// TwinCAT 3 PLC project SampleWeighing
// ProgramVersion: 3.1.4026.20
// libraries:
//   Tc2_Standard, * (Beckhoff Automation GmbH)
//   Tc2_SUPS, * (Beckhoff Automation GmbH)
//   Tc2_System, * (Beckhoff Automation GmbH)
//   Tc2_Utilities, * (Beckhoff Automation GmbH)
//   Tc3_EventLogger, * (Beckhoff Automation GmbH)
//   Tc3_Filter, * (Beckhoff Automation GmbH)
//   Tc3_Module, * (Beckhoff Automation GmbH)
//   Tc3_Weighing, * (Beckhoff Automation GmbH)
// project tree:
//   DUTs/ E_DistributionType.TcDUT (not stored), E_FilterType.TcDUT, E_FunctionType.TcDUT, ST_POINTS.TcDUT
//   GVLs/ Global_Constants.TcGVL, GVL_IO.TcGVL, GVL_WEIGHING_HMI.TcGVL
//   / PlcTask.TcTTO
//   POUs/FBs/ FB_CLOCK.TcPOU (not stored), FB_Filter.TcPOU, FB_Filter59.TcPOU, P_TextModeWrite.TcPOU
//   POUs/ FB_DynamicWeighing.TcPOU, FB_STATS.TcPOU, MAIN.TcPOU, P_HMI.TcPOU, P_LightTest.TcPOU (not stored)
//   POUs/Utilities/ FB_FunctionGenerator.TcPOU
//   VISUs/ RecipeManager.TcRMO (not stored)
// real-time tasks:
//   TASK PlcTask: cycle T#1ms, priority 4, ADS port 350
// I/O:
//   DEVICE Device 2 (EtherCAT), AmsNetId 10.199.162.27.3.1
//     Term 1 (EK1100) [EK1100 EtherCAT Coupler (2A E-Bus)]
//       Term 2 (EL1809) [EL1809 16Ch. Dig. Input 24V, 3ms]
//       Term 3 (EL2808) [EL2808 8Ch. Dig. Output 24V, 0.5A]
//       Term 5 (EL4132)
//       Term 10 (EL9510) [EL9510 Power supply terminal 10V]
//       Term 11 (EL3102) [EL3102 2Ch. Ana. Input +/-10V, Diff.]
//       Term 16 (EL6751) [EL6751 CANopen Master]
//       Term 9 (EL9011) [EL9011 End Terminal]
//     Term 14 (EK1100) [EK1100 EtherCAT Coupler (2A E-Bus)]
//       Term 15 (EL3356-0010) [EL3356-0010 1Ch. Ana. Input Resistor Bridge Terminal, 24bit, High Precision]
//       Term 12 (EL3356) [EL3356 1Ch. Ana. Input Resistor Bridge Terminal, 16bit, High Precision]
//       Term 20 (EK1110) [EK1110 EtherCAT extension]
// variable links:
//   SampleWeighing/SampleWeighing Instance <-> Device 2 (EtherCAT)/Term 1 (EK1100)/Term 2 (EL1809)
//     PlcTask Inputs/GVL_IO.arrDIs[{1..16}] <-> Channel {1..16}/Input  (16 links)
//   SampleWeighing/SampleWeighing Instance <-> Device 2 (EtherCAT)/Term 1 (EK1100)/Term 3 (EL2808)
//     PlcTask Outputs/GVL_IO.arrDOs[{1..8}] <-> Channel {1..8}/Output  (8 links)
//   SampleWeighing/SampleWeighing Instance <-> Device 2 (EtherCAT)/Term 1 (EK1100)/Term 5 (EL4132)
//     PlcTask Outputs/GVL_IO.arrAOs[1] <-> Channel 1/Output
//     PlcTask Outputs/GVL_IO.arrAOs[2] <-> Channel 2/Output
//   SampleWeighing/SampleWeighing Instance <-> Device 2 (EtherCAT)/Term 14 (EK1100)/Term 15 (EL3356-0010)
//     PlcTask Inputs/GVL_IO.EL3356_RawInput <-> RMB Value (Real)/Value (Real)
//     PlcTask Outputs/GVL_IO.EL3356_SampleMode <-> RMB Control/Ctrl/Sample mode

CONFIGURATION SampleWeighing
    RESOURCE PLC ON TwinCAT3
        TASK PlcTask(INTERVAL := T#1ms, PRIORITY := 4);
        PROGRAM MAIN WITH PlcTask : MAIN;
    END_RESOURCE
END_CONFIGURATION

// ---- DUTs/E_FilterType.TcDUT
{attribute 'qualified_only'}
{attribute 'strict'}
{attribute 'to_string'}
TYPE E_FilterType :
(	
	Disabled := 0,
	PTn,
	MovingAverage
);
END_TYPE

// ---- DUTs/E_FunctionType.TcDUT
TYPE E_FunctionType :
(
	eConst := 0,
	eSine,
	eSquare,
	ePulse,
	eTriangular,
	eSawtooth,
	eAM,
	eRand,
	eTrapezoid
);
END_TYPE

// ---- DUTs/ST_POINTS.TcDUT
TYPE ST_POINTS :
STRUCT
	x : REAL;
	y : REAL;
END_STRUCT
END_TYPE

// ---- GVLs/Global_Constants.TcGVL
VAR_GLOBAL CONSTANT
	cOversamples	: UINT := 1;					// number of oversamples
	cSamplingRate	: UINT := 1000 * cOversamples;	// samplerate
END_VAR

// ---- GVLs/GVL_IO.TcGVL
{attribute 'qualified_only'}
VAR_GLOBAL
	arrDIs				 		AT %I*	: ARRAY[1..16] OF BOOL;
	arrDOs			 			AT %Q*	: ARRAY[1..8] OF BOOL;
	arrAIs						AT %I*	: ARRAY[1..2] OF INT;
	arrAOs						AT %Q*	: ARRAY[1..2] OF INT;
	EL3356_RawInput 			AT %I*	: REAL;
	EL3356_SampleMode			AT %Q*	: BOOL := FALSE;
END_VAR

// ---- GVLs/GVL_WEIGHING_HMI.TcGVL
{attribute 'qualified_only'}
VAR_GLOBAL PERSISTENT
	(* Combo Filter Cfg *)
	nFilterOrder 		: UINT := 6;
	rCutOff		 		: REAL	:= 10.0;
	cSamplingRate		: UINT := 100 * cOversamples;	// samplerate
	nSamplesToFilter	: UINT := 200;
	bResetFilter		: BOOL;
	fNotchFrequency		: LREAL;
	
	(* Scaling Params *)
	fRawLow 				: REAL := 0.0;
	fReferenceLow 			: REAL := 0.0;
	fRawHigh 				: REAL := 1000.0;
	fReferenceHigh 			: REAL := 100.0;
	nNumCalibrationSamples 	: UDINT := 100;
	
	(* Weighing Params *)
	nWindowLenght 					: UDINT := 100;
	
	nValidationSamplesValidation	: UDINT := 100;
	fThresholdWeightValidation 		: LREAL := 20.0;
	fMaxStdValidation				: LREAL := 5.0;
	fMaxWeightDeviationValidation	: LREAL := 0.0;
	fRelativeWeightLimit			: LREAL := 0.0;
	fActualRelativeWeightLimit		: LREAL := 0.0;
	
	
	nValidationSamplesAutoTare		: UDINT := 100;
	fThresholdWeightAutoTare 		: REAL := 10.0;
	fMaxStdAutoTare					: LREAL := 1.0;
	fMaxWeightDeviationAutoTare		: LREAL := 0.0;
	
		
	(* Booleans to Reconfigure Filters By IHM *)
	bReconfigureFilter 		: BOOL;
	bReconfigureWeighing 	: BOOL;
	
	(* Calibration *)
	fCalibrateReferenceLow 		: LREAL := 0;
	fCalibrateReferenceHigh 	: LREAL := 1000;
	bCalibrateReferenceLow 		: BOOL := FALSE;
	bCalibrateReferenceHigh 	: BOOL := FALSE;
	bApplyCalibration 			: BOOL := FALSE;
	bAcceptCalibration 			: BOOL := TRUE;
	
	(* Tare *)	
	bTare : BOOL := FALSE;
	fMaxTotalTareLimit : LREAL := 40.0; // set error if total taring amount exceeds the limit
	eAutoTareType : E_WG_AutoTareType := E_WG_AutoTareType.eContinously;
	nNumTareSamples 		: UDINT := 100;
	
	(* Filters Cfg *)	
	
	EFilter1			: E_FilterType;
	EFilter2			: E_FilterType;
	EFilter3			: E_FilterType;
	EFilter4			: E_FilterType;
	EFilter5			: E_FilterType;
	
	(* Filter 1 *)
	fc1				 	: LREAL := 3; // Cut Frequency in Hz
	Tfc1			 	: LREAL := (1.0 / (2.0 * PI * fc1)) / SQRT(EXPT(2.0, 1.0 / 1) - 1.0);
	nGainPTn1			: UINT := 1;
	nOrderPTn1			: UINT := 1;
	fSamplingRatePTn1	: UINT := 1000;
	bReconfigurePTn1	: BOOL;
	
	STFilter1_PTn		: ST_FTR_PTn := (fKp:= 1,
										 fT1 := Tfc1,
										 nOrder := nOrderPTn1,
										 fSamplingRate := fSamplingRatePTn1,
										 nOversamples:= 1,
										 nChannels := 1);
	
	fbFilterPTn1 : FB_FTR_PTn := (stConfig:= STFilter1_PTn);
	
	(* Filter 2 *)
	fc2                  : LREAL := 3;
	Tfc2                 : LREAL := (1.0 / (2.0 * PI * fc2)) / SQRT(EXPT(2.0, 1.0 / 1) - 1.0);
	nGainPTn2            : UINT := 1;
	nOrderPTn2           : UINT := 1;
	fSamplingRatePTn2    : UINT := 1000;
	bReconfigurePTn2     : BOOL;
	
	STFilter2_PTn        : ST_FTR_PTn := (
							fKp:= 1,
							fT1 := Tfc2,
							nOrder := nOrderPTn2,
							fSamplingRate := fSamplingRatePTn2,
							nOversamples:= 1,
							nChannels := 1);
	
	fbFilterPTn2 : FB_FTR_PTn := (stConfig:= STFilter2_PTn);
	
	(* Filter 3 *)
	fc3                  : LREAL := 3;
	Tfc3                 : LREAL := (1.0 / (2.0 * PI * fc3)) / SQRT(EXPT(2.0, 1.0 / 1) - 1.0);
	nGainPTn3            : UINT := 1;
	nOrderPTn3           : UINT := 1;
	fSamplingRatePTn3    : UINT := 1000;
	bReconfigurePTn3     : BOOL;
	
	STFilter3_PTn        : ST_FTR_PTn := (
							fKp:= 1,
							fT1 := Tfc3,
							nOrder := nOrderPTn3,
							fSamplingRate := fSamplingRatePTn3,
							nOversamples:= 1,
							nChannels := 1);
	
	fbFilterPTn3 : FB_FTR_PTn := (stConfig:= STFilter3_PTn);
	
	(* Filter 4 *)
	fc4                  : LREAL := 3;
	Tfc4                 : LREAL := (1.0 / (2.0 * PI * fc4)) / SQRT(EXPT(2.0, 1.0 / 1) - 1.0);
	nGainPTn4            : UINT := 1;
	nOrderPTn4           : UINT := 1;
	fSamplingRatePTn4    : UINT := 1000;
	bReconfigurePTn4     : BOOL;
	
	STFilter4_PTn        : ST_FTR_PTn := (
							fKp:= 1,
							fT1 := Tfc4,
							nOrder := nOrderPTn4,
							fSamplingRate := fSamplingRatePTn4,
							nOversamples:= 1,
							nChannels := 1);
	
	fbFilterPTn4 : FB_FTR_PTn := (stConfig:= STFilter4_PTn);
	
	(* Filter 5 *)
	fc5                  : LREAL := 3;
	Tfc5                 : LREAL := (1.0 / (2.0 * PI * fc5)) / SQRT(EXPT(2.0, 1.0 / 1) - 1.0);
	nGainPTn5            : UINT := 1;
	nOrderPTn5           : UINT := 1;
	fSamplingRatePTn5    : UINT := 1000;
	bReconfigurePTn5     : BOOL;
	
	STFilter5_PTn        : ST_FTR_PTn := (
							fKp:= 1,
							fT1 := Tfc5,
							nOrder := nOrderPTn5,
							fSamplingRate := fSamplingRatePTn5,
							nOversamples:= 1,
							nChannels := 1);
	
	fbFilterPTn5 : FB_FTR_PTn := (stConfig:= STFilter5_PTn);
	
	(* Mirror actual values to simplify to user *)
	(* Validation *)
	nActualWindowLenght 					: UDINT;
	nActualValidationSamplesValidation		: UDINT;
	fActualThresholdWeightValidation 		: LREAL;
	fActualMaxStdValidation					: LREAL;
	fActualMaxWeightDeviationValidation		: LREAL;
	
	(* Last and Actual Weigh Values *)
	fWeight 		: LREAL;
	fLastWeight 	: LREAL;
	fStd 			: LREAL;
	fLastStd 		: LREAL;
	
	(* Lib Booleans *)
	bValidMeasurement 	: BOOL;
	bNewResult			: BOOL;
	bCriteria1			: BOOL;
	bCriteria2			: BOOL;
	bCriteria3			: BOOL;
	
	
END_VAR

// ---- POUs/MAIN.TcPOU
PROGRAM MAIN
VAR
	// Test signal generation
	fRawAmplitudeSignal 	: LREAL := 1000;
	fAbsoluteNoise 			: LREAL := 200;
	fFrequency 				: LREAL := 1; 			// Hz		
	fSamplingRate 			: LREAL := TO_LREAL(cSamplingRate);
	fbSignal 				: FB_FunctionGenerator;
	
	aRawInput 				: ARRAY[1..cOversamples] OF LREAL;
	aRawInputNoise 			: ARRAY[1..cOversamples] OF LREAL;	
	aRawSignal	 			: ARRAY[1..cOversamples] OF LREAL;
	
	// Error handling
	nCountErrors 			: UDINT;
	nEventId 				: UDINT;
	sEventClassName 		: T_MaxString;
	sSourcePath 			: T_MaxString;
	eSeverity 				: TcEventSeverity;
	
	// Weighing
	fbDynamicWeighing 		: FB_DynamicWeighing;
	
	
	//Slope
	bActivateSlope 			: BOOL;
	fDeltaWeight 			: LREAL;
	bAddWeight				: BOOL;
	
	// CP67 UPS Persistent Data
	fbUPS				: FB_S_UPS_BAPI;
	
	stParamsFilterIn 	: ST_WG_ComboFilter;
	stParamsScaleIn		: ST_WG_Scaling;
	stParamsWeighingIn	: ST_WG_Weighing;
	
	bInit				: BOOL;
	bSuccess			: BOOL;
	yFiltroEntrada		: LREAL;
	yFiltroSaida		: LREAL;
	yFiltroSaida2		: LREAL;
	yFiltroSaida3		: LREAL;
	yFiltroSaida4		: LREAL;
	yFiltroSaida5		: LREAL;
				
	bSucceed			: BOOL;
	bReset: BOOL;
END_VAR

// Generate inputs FOR simulation
GenerateInputs();

// Increase the weight continuously.
IF bActivateSlope THEN
	AddSlope();
END_IF

// Increase the weight once
IF bAddWeight THEN
	AddWeight();
	bAddWeight := FALSE;
END_IF

// // Call weighing FB
// fbDynamicWeighing(aInput := aRawInputNoise);

actFilterCfg();
actFilterSignal();

(* Filter Params *)
stParamsFilterIn.nOrder 			:= GVL_WEIGHING_HMI.nFilterOrder;
stParamsFilterIn.fCutoff 			:= GVL_WEIGHING_HMI.rCutOff;
stParamsFilterIn.fSamplingRate 		:= TO_LREAL(GVL_WEIGHING_HMI.cSamplingRate);
stParamsFilterIn.nSamplesToFilter 	:= GVL_WEIGHING_HMI.nSamplesToFilter;
stParamsFilterIn.bReset				:= GVL_WEIGHING_HMI.bResetFilter;
stParamsFilterIn.fNotchFrequency	:= GVL_WEIGHING_HMI.fNotchFrequency;


(* Scale Params *)
stParamsScaleIn.fRawLow 				:= GVL_WEIGHING_HMI.fRawLow;
stParamsScaleIn.fReferenceLow 			:= GVL_WEIGHING_HMI.fReferenceLow;
stParamsScaleIn.fRawHigh		 		:= GVL_WEIGHING_HMI.fRawHigh;
stParamsScaleIn.fReferenceHigh			:= GVL_WEIGHING_HMI.fReferenceHigh;


(* Weighing *)
stParamsWeighingIn.nWindowLength						:= GVL_WEIGHING_HMI.nWindowLenght;
stParamsWeighingIn.Validation.nValidationSamples		:= GVL_WEIGHING_HMI.nValidationSamplesValidation;
stParamsWeighingIn.Validation.fThresholdWeight			:= GVL_WEIGHING_HMI.fThresholdWeightValidation;
stParamsWeighingIn.Validation.fMaxStd					:= GVL_WEIGHING_HMI.fMaxStdValidation;
stParamsWeighingIn.Validation.fMaxWeightDeviation		:= GVL_WEIGHING_HMI.fMaxWeightDeviationValidation;
stParamsWeighingIn.Validation.fRelativeWeightLimit		:= GVL_WEIGHING_HMI.fRelativeWeightLimit;


stParamsWeighingIn.AutoTare.nValidationSamples			:= GVL_WEIGHING_HMI.nValidationSamplesAutoTare;
stParamsWeighingIn.AutoTare.fThresholdWeight			:= GVL_WEIGHING_HMI.fThresholdWeightAutoTare;
stParamsWeighingIn.AutoTare.fMaxStd						:= GVL_WEIGHING_HMI.fMaxStdAutoTare;
stParamsWeighingIn.AutoTare.fMaxWeightDeviation			:= GVL_WEIGHING_HMI.fMaxWeightDeviationAutoTare;


(* Controls *)			  


fbDynamicWeighing(aInput := aRawSignal, 
					stParamsComboFilter 		:= stParamsFilterIn,
					stParamsScale 				:= stParamsScaleIn,
					stParamsWeighing 			:= stParamsWeighingIn,
					nNumCalibrationSamples 		:= GVL_WEIGHING_HMI.nNumCalibrationSamples,
					nNumTareSamples 			:= GVL_WEIGHING_HMI.nNumTareSamples,
					bAcceptCalibration			:= GVL_WEIGHING_HMI.bAcceptCalibration,
					fCalibrateReferenceLow 		:= GVL_WEIGHING_HMI.fCalibrateReferenceLow,
					fCalibrateReferenceHigh 	:= GVL_WEIGHING_HMI.fCalibrateReferenceHigh,
					bTare						:= GVL_WEIGHING_HMI.bTare,
					fMaxTotalTareLimit			:= GVL_WEIGHING_HMI.fMaxTotalTareLimit,
					eAutoTareType				:= GVL_WEIGHING_HMI.eAutoTareType,
);
	
// Error handling
IF fbDynamicWeighing.ipResultMessage <> 0 THEN	
	nEventId := fbDynamicWeighing.ipResultMessage.nEventId;
	sSourcePath := fbDynamicWeighing.ipResultMessage.ipSourceInfo.sName;
	eSeverity := fbDynamicWeighing.ipResultMessage.eSeverity;	
	fbDynamicWeighing.ipResultMessage.RequestEventClassName(1033, sEventClassName, SIZEOF(sEventClassName));
END_IF

IF fbDynamicWeighing.bError THEN
	nCountErrors := nCountErrors + 1;
END_IF


(* HMI Mirroring important variables to user *)
P_HMI();


(* CSV Export *)
//P_TextModeWrite.database();

ACTION actAux:
(* Light Test *)
P_LightTest();

(* HMI *)
P_HMI();

(* UPS *)
fbUPS(
	sNetID:= '', 
	iPLCPort:= 851, 
	tTimeout:= , 
	eUpsMode:= , 
	ePersistentMode:= , 
	tRecoverTime:= , 
	bPowerFailDetect=> , 
	eState=> , 
	nCapacity=> , 
	bBusy=> , 
	bError=> , 
	nErrID=> );
END_ACTION

ACTION actFilterCfg:
IF GVL_WEIGHING_HMI.bReconfigurePTn1 THEN
	GVL_WEIGHING_HMI.STFilter1_PTn.fKp 				:= GVL_WEIGHING_HMI.nGainPTn1;
	GVL_WEIGHING_HMI.STFilter1_PTn.fT1 				:= GVL_WEIGHING_HMI.Tfc1;
	GVL_WEIGHING_HMI.STFilter1_PTn.nOrder 			:= GVL_WEIGHING_HMI.nOrderPTn1;
	GVL_WEIGHING_HMI.STFilter1_PTn.fSamplingRate 	:= GVL_WEIGHING_HMI.fSamplingRatePTn1;
	GVL_WEIGHING_HMI.STFilter1_PTn.nOversamples		:= 1;
	GVL_WEIGHING_HMI.STFilter1_PTn.nChannels 		:= 1;	

	bSuccess := GVL_WEIGHING_HMI.fbFilterPTn1.Configure(stConfig:=GVL_WEIGHING_HMI.STFilter1_PTn);
END_IF


IF bReset THEN
	GVL_WEIGHING_HMI.fbFilterPTn1.Reset();
END_IF


IF GVL_WEIGHING_HMI.bReconfigurePTn2 THEN
	GVL_WEIGHING_HMI.STFilter2_PTn.fKp 				:= GVL_WEIGHING_HMI.nGainPTn2;
	GVL_WEIGHING_HMI.STFilter2_PTn.fT1 				:= GVL_WEIGHING_HMI.Tfc2;
	GVL_WEIGHING_HMI.STFilter2_PTn.nOrder 			:= GVL_WEIGHING_HMI.nOrderPTn2;
	GVL_WEIGHING_HMI.STFilter2_PTn.fSamplingRate 	:= GVL_WEIGHING_HMI.fSamplingRatePTn2;
	GVL_WEIGHING_HMI.STFilter2_PTn.nOversamples		:= 1;
	GVL_WEIGHING_HMI.STFilter2_PTn.nChannels 		:= 1;	

	bSuccess := GVL_WEIGHING_HMI.fbFilterPTn2.Configure(stConfig:=GVL_WEIGHING_HMI.STFilter2_PTn);
END_IF

IF GVL_WEIGHING_HMI.bReconfigurePTn3 THEN
	GVL_WEIGHING_HMI.STFilter3_PTn.fKp 				:= GVL_WEIGHING_HMI.nGainPTn3;
	GVL_WEIGHING_HMI.STFilter3_PTn.fT1 				:= GVL_WEIGHING_HMI.Tfc3;
	GVL_WEIGHING_HMI.STFilter3_PTn.nOrder 			:= GVL_WEIGHING_HMI.nOrderPTn3;
	GVL_WEIGHING_HMI.STFilter3_PTn.fSamplingRate 	:= GVL_WEIGHING_HMI.fSamplingRatePTn3;
	GVL_WEIGHING_HMI.STFilter3_PTn.nOversamples		:= 1;
	GVL_WEIGHING_HMI.STFilter3_PTn.nChannels 		:= 1;	

	bSuccess := GVL_WEIGHING_HMI.fbFilterPTn3.Configure(stConfig:=GVL_WEIGHING_HMI.STFilter3_PTn);
END_IF


IF GVL_WEIGHING_HMI.bReconfigurePTn4 THEN
	GVL_WEIGHING_HMI.STFilter4_PTn.fKp 				:= GVL_WEIGHING_HMI.nGainPTn4;
	GVL_WEIGHING_HMI.STFilter4_PTn.fT1 				:= GVL_WEIGHING_HMI.Tfc4;
	GVL_WEIGHING_HMI.STFilter4_PTn.nOrder 			:= GVL_WEIGHING_HMI.nOrderPTn4;
	GVL_WEIGHING_HMI.STFilter4_PTn.fSamplingRate 	:= GVL_WEIGHING_HMI.fSamplingRatePTn4;
	GVL_WEIGHING_HMI.STFilter4_PTn.nOversamples		:= 1;
	GVL_WEIGHING_HMI.STFilter4_PTn.nChannels 		:= 1;	

	bSuccess := GVL_WEIGHING_HMI.fbFilterPTn4.Configure(stConfig:=GVL_WEIGHING_HMI.STFilter4_PTn);
END_IF


IF GVL_WEIGHING_HMI.bReconfigurePTn5 THEN
	GVL_WEIGHING_HMI.STFilter5_PTn.fKp 				:= GVL_WEIGHING_HMI.nGainPTn5;
	GVL_WEIGHING_HMI.STFilter5_PTn.fT1 				:= GVL_WEIGHING_HMI.Tfc5;
	GVL_WEIGHING_HMI.STFilter5_PTn.nOrder 			:= GVL_WEIGHING_HMI.nOrderPTn5;
	GVL_WEIGHING_HMI.STFilter5_PTn.fSamplingRate 	:= GVL_WEIGHING_HMI.fSamplingRatePTn5;
	GVL_WEIGHING_HMI.STFilter5_PTn.nOversamples		:= 1;
	GVL_WEIGHING_HMI.STFilter5_PTn.nChannels 		:= 1;	

	bSuccess := GVL_WEIGHING_HMI.fbFilterPTn5.Configure(stConfig:=GVL_WEIGHING_HMI.STFilter5_PTn);
END_IF
END_ACTION

ACTION actFilterSignal:
// aRawSignal[1] := GVL_IO.EL3356_RawInput;

// yFiltroEntrada := GVL_IO.EL3356_RawInput;

yFiltroEntrada := aRawInputNoise[1];

(* First Filter *)
IF GVL_WEIGHING_HMI.EFilter1 = 0 THEN // Disabled
	yFiltroSaida := yFiltroEntrada;	
ELSIF GVL_WEIGHING_HMI.EFilter1 = 1 THEN // PTn
	bSucceed := GVL_WEIGHING_HMI.fbFilterPTn1.Call(ADR(yFiltroEntrada), SIZEOF(yFiltroEntrada), ADR(yFiltroSaida), SIZEOF(yFiltroSaida));
END_IF

(* Second Filter *)
IF GVL_WEIGHING_HMI.EFilter2 = 0 THEN // Disabled
	yFiltroSaida2 := yFiltroSaida;	
ELSIF GVL_WEIGHING_HMI.EFilter2 = 1 THEN // PTn
	bSucceed := GVL_WEIGHING_HMI.fbFilterPTn2.Call(ADR(yFiltroSaida), SIZEOF(yFiltroSaida), ADR(yFiltroSaida2), SIZEOF(yFiltroSaida2));
END_IF

(* Third Filter *)
IF GVL_WEIGHING_HMI.EFilter3 = 0 THEN // Disabled
	yFiltroSaida3 := yFiltroSaida2;	
ELSIF GVL_WEIGHING_HMI.EFilter3 = 1 THEN // PTn
	bSucceed := GVL_WEIGHING_HMI.fbFilterPTn2.Call(ADR(yFiltroSaida2), SIZEOF(yFiltroSaida2), ADR(yFiltroSaida3), SIZEOF(yFiltroSaida3));
END_IF

(* Fourth Filter *)
IF GVL_WEIGHING_HMI.EFilter4 = 0 THEN // Disabled
	yFiltroSaida4 := yFiltroSaida3;	
ELSIF GVL_WEIGHING_HMI.EFilter4 = 1 THEN // PTn
	bSucceed := GVL_WEIGHING_HMI.fbFilterPTn2.Call(ADR(yFiltroSaida3), SIZEOF(yFiltroSaida3), ADR(yFiltroSaida4), SIZEOF(yFiltroSaida4));
END_IF

(* Fifth Filter *)
IF GVL_WEIGHING_HMI.EFilter5 = 0 THEN // Disabled
	yFiltroSaida5 := yFiltroSaida4;	
ELSIF GVL_WEIGHING_HMI.EFilter5 = 1 THEN // PTn
	bSucceed := GVL_WEIGHING_HMI.fbFilterPTn2.Call(ADR(yFiltroSaida4), SIZEOF(yFiltroSaida4), ADR(yFiltroSaida5), SIZEOF(yFiltroSaida5));
END_IF


aRawSignal[1] := yFiltroSaida5; // Recebe sempre a última saída
END_ACTION

METHOD AddSlope : BOOL
VAR_INPUT
END_VAR
VAR
	idx : UINT;
	fSlope: LREAL := 0.2;
END_VAR
fDeltaWeight := fDeltaWeight + fSlope;
END_METHOD

METHOD AddWeight : BOOL
VAR_INPUT
END_VAR
VAR
	idx : UINT;
	fAddWeight: LREAL := 100;
END_VAR
fDeltaWeight := fDeltaWeight + fAddWeight;
END_METHOD

METHOD GenerateInputs : BOOL
VAR_INPUT
END_VAR
VAR
	idx : UINT;
END_VAR
fbSignal(				
	fSamplingRate := fSamplingRate,
	nOversamples := cOversamples,
	fFrequency := fFrequency,
	fAmplitude := 2.0 * fRawAmplitudeSignal,
	eFunction := E_FunctionType.eTrapezoid,							
	aSignal => aRawInput);


FOR idx := 1 TO cOversamples DO
	aRawInput[idx] := aRawInput[idx] + fDeltaWeight;
END_FOR		 

MEMCPY(ADR(aRawInputNoise),ADR(aRawInput),SIZEOF(aRawInputNoise));
fbSignal.AddAbsoluteNoise(fAbsoluteNoise, aRawInputNoise);
END_METHOD

END_PROGRAM

// ---- POUs/Utilities/FB_FunctionGenerator.TcPOU
// generates a signal build up by the specified function type. v1.4
// generates random signal (uniform, normal or chi-squared)

FUNCTION_BLOCK FB_FunctionGenerator
VAR_INPUT
	bEnable		: BOOL 	:= TRUE;
	fSamplingRate : LREAL := 10000.0; // in Hz
	nOversamples : UDINT := 10;
	fFrequency	: LREAL := 1000;	// in [Hz]
	fAmplitude	: LREAL := 1;
	fOffset		: LREAL	:= 0;	
	nDutyCycle	: UINT 	:= 50;		// % (for pulse function)
	nSeed		: INT	:= 1;	 
	aRange		: ARRAY [1..2] OF LREAL := [0,1];
	eRandType	: E_DistributionType	:= E_DistributionType.eNormal;
	eFunction	: E_FunctionType := E_FunctionType.eSine;	
END_VAR
VAR_OUTPUT
	bError		: BOOL;
	aSignal		: ARRAY[1..cOversamples] OF LREAL;
END_VAR
VAR
	bInit						: BOOL := TRUE;
	fLastSamplingRate : LREAL;
	nLastOversamples : UDINT;
	fLastFrequency				: LREAL;		// in [Hz]
	fLastAmplitude				: LREAL;
	fLastOffset					: LREAL;
	nLastDutyCycle				: UINT;
	eLastFunction				: E_FunctionType;
	
	nSamples					: UDINT;
	fCycleTime					: LREAL;		// in [s]
	fDelta						: LREAL;		// amplitude delta per sample
	fPhase						: LREAL;		// in [°]
	nSign						: INT := 1;		// 1 or -1
	fLastSignalValue			: LREAL;		// amplitude
	fPeriod						: LREAL;		// in [s]
	fAngularIncrement			: LREAL;		// in [°]
	fAngularIncrementPerCycle	: LREAL;		// in [°]
	fAngularIncrementPerSample	: LREAL;		// in [°]
	(* for modulated signal *)
	fCarrierFrequency			: LREAL := 500;	// in [Hz] (sine)
	fCarrierAmplitude			: LREAL := 1;
	fCarrierPeriod				: LREAL;		// in [s]
	fCarrierAngularIncrement			: LREAL;		// in [°]
	fCarrierAngularIncrementPerCycle	: LREAL;		// in [°]
	fCarrierAngularIncrementPerSample	: LREAL;		// in [°]
	
	fbDrand						: ARRAY[1..cOversamples] OF DRAND;		
	bNormalDist					: BOOL := TRUE;
	
	fY1							: LREAL;
	fY2							: LREAL;
	fX1							: LREAL;
	fX2							: LREAL;
	
	fbRAND1						: DRAND;
	fbRAND2						: DRAND;				
END_VAR

IF bEnable THEN

	IF fLastSamplingRate <> fSamplingRate THEN
		bInit := TRUE; // For automatic initializing
		fLastSamplingRate := fSamplingRate;
	END_IF
	IF nLastOversamples <> nOversamples THEN
		bInit := TRUE; // For automatic initializing
		nLastOversamples := nOversamples;
	END_IF
	
	IF fLastFrequency <> fFrequency THEN
		bInit := TRUE; // For automatic initializing
		fLastFrequency := fFrequency;
	END_IF
	IF fLastAmplitude <> fAmplitude THEN
		bInit := TRUE; // For automatic initializing
		fLastAmplitude := fAmplitude;
	END_IF
	IF fLastOffset <> fOffset THEN
		bInit := TRUE; // For automatic initializing
		fLastOffset := fOffset;
	END_IF
	IF nLastDutyCycle <> nDutyCycle THEN
		bInit := TRUE; // For automatic initializing
		nLastDutyCycle := nDutyCycle;
	END_IF
	IF eLastFunction <> eFunction THEN
		bInit := TRUE; // For automatic initializing
		eLastFunction := eFunction;
	END_IF
	IF bInit THEN
		// Get taks info	
//		fbGetTaskIdx();
//		fCycleTime := TwinCAT_SystemInfoVarList._TaskInfo[fbGetTaskIdx.index].CycleTime (*100ns*) / (10.0 * 1000.0 * 1000.0);	
		fCycleTime	 := nOversamples/fSamplingRate;
		fLastSignalValue := 0;
		nSign := 1;
		fAngularIncrement := 0;
		// Flush out old data
		MEMSET(ADR(aSignal), 0, SIZEOF(aSignal));
		IF fFrequency <> 0 AND fCycleTime > 0 THEN		
			// Calculate period, increments per plc cycle, increment per oversample
			IF cOversamples <> 0 THEN			
				IF eFunction = E_FunctionType.eSine THEN
					fPeriod := 1/fFrequency;
					fAngularIncrementPerCycle := 360*(fCycleTime/fPeriod);
					fAngularIncrementPerSample := fAngularIncrementPerCycle/cOversamples;
					// no phase adjustment
					bInit := FALSE;
				ELSIF eFunction = E_FunctionType.eConst	THEN
					bInit := FALSE;	
				ELSIF eFunction = E_FunctionType.eSquare	THEN
					fPeriod := 1/fFrequency;
					fAngularIncrementPerCycle := 360*(fCycleTime/fPeriod);
					fAngularIncrementPerSample := fAngularIncrementPerCycle/cOversamples;
					fPhase := 0.5*360;
					bInit := FALSE;
				ELSIF eFunction = E_FunctionType.ePulse THEN
					fPeriod := 1/fFrequency;
					fAngularIncrementPerCycle := 360*(fCycleTime/fPeriod);
					fAngularIncrementPerSample := fAngularIncrementPerCycle/cOversamples;
					IF nDutyCycle > 100 THEN
						nDutyCycle := 100;
					END_IF
					fPhase := (UDINT_TO_LREAL(nDutyCycle)/100)*360;
					bInit := FALSE;					
				ELSIF eFunction = E_FunctionType.eTriangular THEN
					fPeriod := 1/fFrequency;				
					fAngularIncrementPerCycle := 360*(fCycleTime/fPeriod);
					fAngularIncrementPerSample := fAngularIncrementPerCycle/cOversamples;
					fPhase := 0.5*360; 
					fDelta := 4*(fAmplitude/(360/fAngularIncrementPerSample));				
					bInit := FALSE;
				ELSIF eFunction = E_FunctionType.eTrapezoid THEN
					fPeriod := 1/fFrequency;				
					fAngularIncrementPerCycle := 360*(fCycleTime/fPeriod);
					fAngularIncrementPerSample := fAngularIncrementPerCycle/cOversamples;
					fPhase := 0.5*360; 
					fDelta := 4*(fAmplitude/(360/fAngularIncrementPerSample));				
					bInit := FALSE;					
				ELSIF eFunction = E_FunctionType.eSawtooth THEN
					fPeriod := 1/fFrequency;			
					fAngularIncrementPerCycle := 360*(fCycleTime/fPeriod);		
					fAngularIncrementPerSample := fAngularIncrementPerCycle/cOversamples;
					fDelta := fAmplitude/(360/fAngularIncrementPerSample);
					bInit := FALSE;
				ELSIF eFunction = E_FunctionType.eAM THEN
					fPeriod := 1/fFrequency;
					fAngularIncrementPerCycle := 360*(fCycleTime/fPeriod);
					fAngularIncrementPerSample := fAngularIncrementPerCycle/cOversamples;
					// no phase adjustment
					fCarrierPeriod := 1/fCarrierFrequency;
					fCarrierAngularIncrementPerCycle := 360*(fCycleTime/fCarrierPeriod);
					fCarrierAngularIncrementPerSample := fCarrierAngularIncrementPerCycle/cOversamples;				
					// no phase adjustment	
					bInit := FALSE;			
				ELSIF eFunction = E_FunctionType.eRand THEN	
					fbRAND1(Seed := nSeed);
					fbRAND2(Seed := nSeed+1);
					bInit := FALSE;
				ELSE
					bError := TRUE;	
				END_IF
			ELSE
				bError := TRUE;
			END_IF
		ELSE
			bError := TRUE;
		END_IF
	END_IF
	
	// Enable function generator
	IF NOT bError THEN		
		CASE eFunction OF		
			// const: constant signal
			E_FunctionType.eConst: Const();
			
			// sine: typical for vibrations originating from rotating machine
			E_FunctionType.eSine: Sine();			
			
			// square: mixed sine signals good for analyzing spectrum				
			E_FunctionType.eSquare: Square();
			
			// pulse: mixed sine signals good for analyzing spectrum				
			E_FunctionType.ePulse: Pulse();
	
			// sawtooth: ramp-type vibrations, continuously increasing			
			E_FunctionType.eSawtooth: Sawtooth();
		
			// triangular: mixed sine signals good for analyzing spectrum
			E_FunctionType.eTriangular: Triangular();
			
			// Trapezoid: trapezoid signal
			E_FunctionType.eTrapezoid: Trapezoid();
		
			// amplitude modulation: typical for vibrations originating from gear-tooth failure or bearing faults
			// Carrier signal with own frequency and amplitude		
			E_FunctionType.eAM: AM();	

			// random nosie: typical for disturbance signal				
		END_CASE
	END_IF
ELSE
	// Flush out old data
	MEMSET(ADR(aSignal), 0, SIZEOF(aSignal));
END_IF

METHOD PUBLIC AddAbsoluteNoise
VAR_INPUT
	fAbsoluteNoise	: LREAL;
END_VAR
VAR_IN_OUT
	aSignal		: ARRAY[1..cOversamples] OF LREAL;
END_VAR
VAR
	fNoise :LREAL;
END_VAR
FOR nSamples := 1 TO cOversamples DO	
	fbRAND1(Num => fNoise); // betwenn 0-1
	fNoise:= (fNoise*2 -1.0) * fAbsoluteNoise;
	aSignal[nSamples] := aSignal[nSamples] + fNoise;
END_FOR
END_METHOD

METHOD PRIVATE AM
VAR_INPUT
END_VAR
FOR nSamples := 1 TO cOversamples DO
	// base signal * carrier signal
	aSignal[nSamples] := ( fAmplitude*SIN(2*PI*(fAngularIncrement+(nSamples-1)*fAngularIncrementPerSample)/360) + fOffset )
							* ( fCarrierAmplitude*SIN(2*PI*(fCarrierAngularIncrement+(nSamples-1)*fCarrierAngularIncrementPerSample)/360) );
END_FOR
// Increment angular positions
fAngularIncrement := fAngularIncrement + fAngularIncrementPerCycle;
fCarrierAngularIncrement := fCarrierAngularIncrement + fCarrierAngularIncrementPerCycle;
END_METHOD

METHOD PRIVATE Const
VAR_INPUT
END_VAR
FOR nSamples := 1 TO cOversamples DO
	
	aSignal[nSamples] := fAmplitude;
	
	aSignal[nSamples] := aSignal[nSamples] + fOffset;
END_FOR
END_METHOD

METHOD PRIVATE Pulse
VAR_INPUT
END_VAR
FOR nSamples := 1 TO cOversamples DO
	// For pulse wave (unequal phases)
	IF (fAngularIncrement >= 360) THEN
		fAngularIncrement := fAngularIncrement - DINT_TO_LREAL(LREAL_TO_DINT(fAngularIncrement/360))*360;
		// or with Tc2_Math library: fAngularIncrement := LMOD(fAngularIncrement,360);
	END_IF
	IF (fAngularIncrement < fPhase) THEN
		nSign := 1;		
	ELSIF (fAngularIncrement >= fPhase) THEN
		nSign := 0;
	END_IF
	fAngularIncrement := fAngularIncrement + fAngularIncrementPerSample;
	
	aSignal[nSamples] := nSign*fAmplitude;
	
	aSignal[nSamples] := aSignal[nSamples] + fOffset;
END_FOR
END_METHOD

METHOD PRIVATE Sawtooth
VAR_INPUT
END_VAR
FOR nSamples := 1 TO cOversamples DO
	// For sawtooth wave (equal phase = period/2)
	IF (fAngularIncrement >= 360) THEN
		fAngularIncrement := fAngularIncrement - DINT_TO_LREAL(LREAL_TO_DINT(fAngularIncrement/360))*360;
		// or with Tc2_Math library: fAngularIncrement := LMOD(fAngularIncrement,360);
		fLastSignalValue := fLastSignalValue -fAmplitude;
	END_IF
	fAngularIncrement := fAngularIncrement + fAngularIncrementPerSample;

	aSignal[nSamples] := fLastSignalValue + fDelta;

	// Store last sample
	fLastSignalValue := aSignal[nSamples];
	
	aSignal[nSamples] := aSignal[nSamples] + fOffset;					
END_FOR
END_METHOD

METHOD PRIVATE Sine
VAR_INPUT
END_VAR
FOR nSamples := 1 TO cOversamples DO
	aSignal[nSamples] := fAmplitude*SIN(2*PI*(fAngularIncrement+(nSamples-1)*fAngularIncrementPerSample)/360);

	aSignal[nSamples] := aSignal[nSamples] + fOffset;
END_FOR

// Increment angular position
fAngularIncrement := fAngularIncrement + fAngularIncrementPerCycle;
END_METHOD

METHOD PRIVATE Square
VAR_INPUT
END_VAR
FOR nSamples := 1 TO cOversamples DO
	// For square wave (equal phase = period/2)
	IF (fAngularIncrement >= 360) THEN
		fAngularIncrement := fAngularIncrement - DINT_TO_LREAL(LREAL_TO_DINT(fAngularIncrement/360))*360;
		// or with Tc2_Math library: fAngularIncrement := LMOD(fAngularIncrement,360);
	END_IF
	IF (fAngularIncrement < fPhase) THEN
		nSign := 1;
	ELSIF (fAngularIncrement >= fPhase) THEN
		nSign := -1;
	END_IF
	fAngularIncrement := fAngularIncrement + fAngularIncrementPerSample;
	
	aSignal[nSamples] := nSign*fAmplitude;
	
	aSignal[nSamples] := aSignal[nSamples] + fOffset;
END_FOR
END_METHOD

METHOD PRIVATE Trapezoid
VAR_INPUT
END_VAR
FOR nSamples := 1 TO cOversamples DO
	IF (fAngularIncrement >= 360) THEN
		fAngularIncrement := fAngularIncrement - DINT_TO_LREAL(LREAL_TO_DINT(fAngularIncrement/360))*360;
		// or with Tc2_Math library: fAngularIncrement := LMOD(fAngularIncrement,360);
	END_IF
	// Negative delta -> Positive delta
	IF fAngularIncrement < fPhase/2 THEN	
		nSign := 1;		
	ELSIF fAngularIncrement >= fPhase/2 AND fAngularIncrement < fPhase THEN
		nSign := -1;
	ELSIF fAngularIncrement >= fPhase THEN
		nSign := 0;	
	END_IF
	fAngularIncrement := fAngularIncrement + fAngularIncrementPerSample;
	
	aSignal[nSamples] := fLastSignalValue + nSign*fDelta;
	IF aSignal[nSamples] > fAmplitude THEN
		aSignal[nSamples] := aSignal[nSamples] - 2*(aSignal[nSamples]-fAmplitude);
	ELSIF aSignal[nSamples] < (-1)*fAmplitude THEN
		aSignal[nSamples] := aSignal[nSamples] - 2*(aSignal[nSamples]+fAmplitude);
	END_IF
	
	// Store last sample
	fLastSignalValue := aSignal[nSamples];		
	
	IF fLastSignalValue > fAmplitude * 0.5 THEN
		aSignal[nSamples] := fAmplitude * 0.5;
	END_IF
	
	aSignal[nSamples] := aSignal[nSamples] + fOffset;
END_FOR
END_METHOD

METHOD PRIVATE Triangular
VAR_INPUT
END_VAR
FOR nSamples := 1 TO cOversamples DO
	IF (fAngularIncrement >= 360) THEN
		fAngularIncrement := fAngularIncrement - DINT_TO_LREAL(LREAL_TO_DINT(fAngularIncrement/360))*360;
		// or with Tc2_Math library: fAngularIncrement := LMOD(fAngularIncrement,360);
	END_IF
	// Negative delta -> Positive delta
	IF fAngularIncrement < fPhase/2 THEN	
		nSign := 1;		
	ELSIF fAngularIncrement >= fPhase/2 AND fAngularIncrement < 3*fPhase/2 THEN
		nSign := -1;
	ELSIF fAngularIncrement >= 3*fPhase/2 THEN
		nSign := 1;	
	END_IF
	fAngularIncrement := fAngularIncrement + fAngularIncrementPerSample;
	
	aSignal[nSamples] := fLastSignalValue + nSign*fDelta;
	IF aSignal[nSamples] > fAmplitude THEN
		aSignal[nSamples] := aSignal[nSamples] - 2*(aSignal[nSamples]-fAmplitude);
	ELSIF aSignal[nSamples] < (-1)*fAmplitude THEN
		aSignal[nSamples] := aSignal[nSamples] - 2*(aSignal[nSamples]+fAmplitude);
	END_IF
	
	// Store last sample
	fLastSignalValue := aSignal[nSamples];		
	
	aSignal[nSamples] := aSignal[nSamples] + fOffset;
END_FOR
END_METHOD

END_FUNCTION_BLOCK

// ---- POUs/FB_DynamicWeighing.TcPOU
FUNCTION_BLOCK FB_DynamicWeighing
VAR_INPUT
	aInput : ARRAY[1..cOversamples] OF LREAL;
	
	// Filter
	stParamsComboFilter 		: ST_WG_ComboFilter;
	
	// Scaling
	stParamsScale 				: ST_WG_Scaling;
	
	// Weighing
	stParamsWeighing 			: ST_WG_Weighing;
	
	// Control
	// Reconfigure
	bReconfigureFilter 			: BOOL := FALSE;
	bReconfigureWeighing 		: BOOL := FALSE;
	
	// Calibration
	nNumCalibrationSamples 		: UDINT := 100;
	fCalibrateReferenceLow 		: LREAL := 417;
	fCalibrateReferenceHigh 	: LREAL := 1215;
	bCalibrateReferenceLow 		: BOOL 	:= FALSE;		// e.g. ref: 417	| raw: 175000
	bCalibrateReferenceHigh 	: BOOL 	:= FALSE;	// e.g. ref: 1215	| raw: 525000	
	bApplyCalibration 			: BOOL 	:= FALSE;
	bAcceptCalibration 			: BOOL 	:= TRUE;
	
	// Tare
	nNumTareSamples 			: UDINT := 100;
	bTare 						: BOOL 	:= FALSE;
	fMaxTotalTareLimit 			: LREAL := 40.0; // set error if total taring amount exceeds the limit
	eAutoTareType 				: E_WG_AutoTareType := E_WG_AutoTareType.eContinously;
	
	
	bDisableFilter				: BOOL;
END_VAR
VAR_OUTPUT
	bError 						: BOOL;
	ipResultMessage 			: I_TcMessage;
	bNewResult 					: BOOL;	
	bValidMeasurement 			: BOOL;	
	fWeight 					: LREAL;
	fLastWeight 				: LREAL;
	fStd 						: LREAL;
	fLastStd 					: LREAL;
	
	(* Extra Diag Values to Show on HMI *)
	(* Validation Values *)
	nActualWindowLenght					: UDINT;
	nActualValidationSamplesValidation	: UDINT;
	fActualThresholdWeightValidation 	: LREAL;
	fActualMaxStdValidation			    : LREAL;
	fActualMaxWeightDeviationValidation : LREAL;
	fActualRelativeWeightLimit			: LREAL;	
	
	fMax : LREAL;
	fMin : LREAL;
END_VAR
VAR
	fbComboFilter 				: FB_WG_ComboFilter	:= (stConfig := stParamsComboFilter);
	fbScale 					: FB_WG_Scaling		:= (stConfig := stParamsScale, eTraceLevel:=TcEventSeverity.Info);
	fbWeighing 					: FB_WG_Weighing	:= (stConfig := stParamsWeighing);
	//					: FB_FTR_PTn(stConfig:= );
	
	
	
	// Helper
	aOutFilter 					: ARRAY[1..cOversamples] OF LREAL; // Stage1 PTn filter, Stage2 MovAvg Filter
	aOutScaling 				: ARRAY[1..cOversamples] OF LREAL; // Scaling
	reconfigureFilter 			: R_TRIG;
	reconfigureWeighing 		: R_TRIG;
	calibrateReferenceLow 		: R_TRIG;
	calibrateReferenceHigh 		: R_TRIG;
	applyCalibration 			: R_TRIG;
	tare 						: R_TRIG;
	

	
	//UserMessage
	fbCustomMessage 	: FB_TcMessage;
	bInit				: BOOL;
	bSucceed			: BOOL;
	
END_VAR

bError := FALSE;
CommandTrigger();
// Configure the FB_WG_Scaling block

IF NOT bInit THEN
	bSucceed := fbScale.Configure(stConfig:=stParamsScale);	
	bInit := TRUE;
END_IF

// Reconfigure
IF reconfigureFilter.Q AND_THEN NOT fbComboFilter.Configure(stParamsComboFilter) THEN
	SetError(fbComboFilter);
END_IF

IF reconfigureWeighing.Q AND_THEN NOT fbWeighing.Configure(stParamsWeighing) THEN
	SetError(fbWeighing);
END_IF

// Calibration	 
IF calibrateReferenceLow.Q AND_THEN NOT fbScale.CalibrateRefLow(nNumCalibrationSamples, fCalibrateReferenceLow) THEN
	SetError(fbScale);
END_IF

IF calibrateReferenceHigh.Q AND_THEN NOT fbScale.CalibrateRefHigh(nNumCalibrationSamples, fCalibrateReferenceHigh) THEN
	SetError(fbScale);
END_IF

IF applyCalibration.Q AND_THEN NOT fbScale.ApplyCalibration(bAcceptCalibration) THEN
	SetError(fbScale);
END_IF

// Tare
IF tare.Q AND_THEN NOT fbScale.Tare(nNumTareSamples) THEN
	SetError(fbScale);
END_IF


// Perform taring process continously if fbWeighing.fAutoTareOffset is not zero
// Careful: ST_WG_Weighing_AutoTare.nValidationSamples should be large enough, to find the best tare weight.
// Execute AutoTare
IF NOT fbWeighing.AutoTare(fbScale, eAutoTareType)THEN
	SetError(fbWeighing);
END_IF

IF ABS(fbScale.fCurrentTareOffset - fbWeighing.fAutoTareOffset) > fMaxTotalTareLimit THEN
	SetCustomWarning(fbCustomMessage, 'Total taring amount exceeds the limit. Please check the weighing machine!');
END_IF


// Execute weighing
IF NOT bDisableFilter THEN
	IF NOT fbComboFilter.Call(ADR(aInput), SIZEOF(aInput), ADR(aOutFilter), SIZEOF(aOutFilter)) THEN
		SetError(fbComboFilter);
	END_IF
ELSE
	aOutFilter := aInput;
END_IF

IF NOT fbScale.Call(ADR(aOutFilter), SIZEOF(aOutFilter), ADR(aOutScaling), SIZEOF(aOutScaling)) THEN
	SetError(fbScale);
END_IF

IF NOT fbWeighing.Call(ADR(aOutScaling), SIZEOF(aOutScaling)) THEN
	SetError(fbWeighing);
END_IF

// Assign results
AssignResults();

// Assign diag values
AssignDiagValues();

METHOD AssignDiagValues : BOOL
VAR_INPUT
END_VAR
(* Actual fbWeighing Block Cfg *)
nActualWindowLenght 					:= fbWeighing.stConfig.nWindowLength;
nActualValidationSamplesValidation		:= fbWeighing.stConfig.Validation.nValidationSamples;
fActualThresholdWeightValidation 		:= fbWeighing.stConfig.Validation.fThresholdWeight;
fActualMaxStdValidation			    	:= fbWeighing.stConfig.Validation.fMaxStd;
fActualMaxWeightDeviationValidation 	:= fbWeighing.stConfig.Validation.fMaxWeightDeviation;
fActualRelativeWeightLimit				:= fbWeighing.stConfig.Validation.fRelativeWeightLimit;
END_METHOD

METHOD AssignResults : BOOL
VAR_INPUT
END_VAR

VAR_OUTPUT
END_VAR
bNewResult := fbWeighing.bNewResult;	
bValidMeasurement := fbWeighing.bValidMeasurement;	
fWeight := fbWeighing.fWeight;
fLastWeight := fbWeighing.fLastWeight;
fStd := fbWeighing.fStd;
fLastStd := fbWeighing.fLastStd;

fMax := fbWeighing.fMax;
fMin := fbWeighing.fMin;
END_METHOD

METHOD CommandTrigger : BOOL
VAR_INPUT
END_VAR
reconfigureFilter(CLK:=bReconfigureFilter OR GVL_WEIGHING_HMI.bReconfigureFilter);
reconfigureWeighing(CLK:=bReconfigureWeighing OR GVL_WEIGHING_HMI.bReconfigureWeighing);
calibrateReferenceLow(CLK:=bCalibrateReferenceLow OR GVL_WEIGHING_HMI.bCalibrateReferenceLow);
calibrateReferenceHigh(CLK:=bCalibrateReferenceHigh OR GVL_WEIGHING_HMI.bCalibrateReferenceHigh);
applyCalibration(CLK:=bApplyCalibration OR GVL_WEIGHING_HMI.bApplyCalibration);
tare(CLK:=bTare);
END_METHOD

METHOD SetCustomWarning : BOOL
VAR_INPUT
	fb : REFERENCE TO FB_TcMessage;
	sText : STRING;
END_VAR
VAR
END_VAR
THIS^.bError := TRUE;
fb.CreateEx(TC_EVENTS.TcWeighingEventClass.Warning_InvalidThreshold,0);
fb.ipArguments.Clear();
fb.ipArguments.AddString(sText);
fb.Send(0);
THIS^.ipResultMessage := fb;
END_METHOD

METHOD SetError : BOOL
VAR_INPUT
	fb : REFERENCE TO _FB_WG_BasicImplementationAlgorithm;
END_VAR
THIS^.bError := fb.bError;
THIS^.ipResultMessage := fb.ipResultMessage;
END_METHOD

END_FUNCTION_BLOCK

// ---- POUs/P_HMI.TcPOU
PROGRAM P_HMI
VAR
	fDelta: LREAL;
END_VAR

(* Actual Validation Values on FB_WEIGHING Block*)

GVL_WEIGHING_HMI.nActualWindowLenght 					 	:= MAIN.fbDynamicWeighing.stParamsWeighing.nWindowLength;

GVL_WEIGHING_HMI.nActualWindowLenght 					 	:= MAIN.fbDynamicWeighing.nActualWindowLenght;
GVL_WEIGHING_HMI.nActualValidationSamplesValidation		 	:= MAIN.fbDynamicWeighing.nActualValidationSamplesValidation;
GVL_WEIGHING_HMI.fActualThresholdWeightValidation 		 	:= MAIN.fbDynamicWeighing.fActualThresholdWeightValidation;
GVL_WEIGHING_HMI.fActualMaxStdValidation					:= MAIN.fbDynamicWeighing.fActualMaxStdValidation;
GVL_WEIGHING_HMI.fActualMaxWeightDeviationValidation		:= MAIN.fbDynamicWeighing.fActualMaxWeightDeviationValidation;
GVL_WEIGHING_HMI.fActualRelativeWeightLimit					:= MAIN.fbDynamicWeighing.fActualRelativeWeightLimit;

GVL_WEIGHING_HMI.fWeight 									:= MAIN.fbDynamicWeighing.fWeight;
GVL_WEIGHING_HMI.fLastWeight 								:= MAIN.fbDynamicWeighing.fLastWeight;
GVL_WEIGHING_HMI.fStd 										:= MAIN.fbDynamicWeighing.fStd;
GVL_WEIGHING_HMI.fLastStd 									:= MAIN.fbDynamicWeighing.fLastStd;


(* Booleans *)

GVL_WEIGHING_HMI.bValidMeasurement 	:= MAIN.fbDynamicWeighing.bValidMeasurement;
GVL_WEIGHING_HMI.bNewResult			:= MAIN.fbDynamicWeighing.bNewResult;

(* Auto Reset Reconfigure Bits *)
IF GVL_WEIGHING_HMI.bReconfigureWeighing THEN
	GVL_WEIGHING_HMI.bReconfigureWeighing := FALSE;
END_IF


(* Bit for Criterias Management *)
IF MAIN.fbDynamicWeighing.fWeight > MAIN.fbDynamicWeighing.fActualThresholdWeightValidation THEN
	GVL_WEIGHING_HMI.bCriteria1 := TRUE;
	fDelta := MAIN.fbDynamicWeighing.fMax - MAIN.fbDynamicWeighing.fMin;	
	IF MAIN.fbDynamicWeighing.fMax - MAIN.fbDynamicWeighing.fMin 
		< MAIN.fbDynamicWeighing.fActualMaxWeightDeviationValidation THEN
			GVL_WEIGHING_HMI.bCriteria2 := TRUE;
		IF MAIN.fbDynamicWeighing.fStd < MAIN.fbDynamicWeighing.fActualMaxStdValidation THEN
			GVL_WEIGHING_HMI.bCriteria3 := TRUE;
		END_IF
	END_IF
ELSE (* Reset everytime weight is < than threshold *)
	GVL_WEIGHING_HMI.bCriteria1 := FALSE;
	GVL_WEIGHING_HMI.bCriteria2 := FALSE;
	GVL_WEIGHING_HMI.bCriteria3	:= FALSE;
END_IF

END_PROGRAM

// ---- POUs/FBs/FB_Filter.TcPOU
FUNCTION_BLOCK FB_Filter
VAR_INPUT
	rEntrada: REAL;
END_VAR
VAR_OUTPUT
	rSaida: REAL;
END_VAR
VAR
	arCoef_Taps10: ARRAY[1..10] OF REAL;
	arLeitura: ARRAY[1..10] OF REAL;
	i: INT;
	rAux: REAL;
END_VAR

//Filtro - FPB_11Hz_10taps

arCoef_Taps10[1] := 	8.84359775738877E-002;
arCoef_Taps10[2] := 	9.59556442767806E-002;
arCoef_Taps10[3] := 	1.01831088400691E-001;
arCoef_Taps10[4] := 	1.05863099175751E-001;
arCoef_Taps10[5] := 	1.07914190572890E-001;
arCoef_Taps10[6] := 	1.07914190572890E-001;
arCoef_Taps10[7] := 	1.05863099175751E-001;
arCoef_Taps10[8] :=		1.01831088400691E-001;
arCoef_Taps10[9] :=		9.59556442767806E-002;
arCoef_Taps10[10] :=	8.84359775738877E-002;

rSaida := 0.0;
FOR i:= 10 TO 2 BY -1 DO
	arLeitura[i] := arLeitura[i-1];	
	rAux := arLeitura[i] * arCoef_Taps10[i];
	rSaida := rSaida + rAux;
END_FOR

arLeitura[1] := rEntrada;

rSaida := rSaida + (arLeitura[1] * arCoef_Taps10[1]);

END_FUNCTION_BLOCK

// ---- POUs/FBs/FB_Filter59.TcPOU
FUNCTION_BLOCK FB_Filter59
VAR_INPUT
	rEntrada: REAL;
END_VAR
VAR_OUTPUT
	rSaida: REAL;
END_VAR
VAR
	arCoef_Taps: ARRAY[1..59] OF REAL;
	arLeitura: ARRAY[1..59] OF REAL;
	i: INT;
	rAux: REAL;
END_VAR

//Fir6 Kaiser - 59Taps


arCoef_Taps[1] := 	1.54135308723898E-002;
arCoef_Taps[2] := 	1.55675060506758E-002;
arCoef_Taps[3] := 	1.57169226616965E-002;
arCoef_Taps[4] := 	1.58616933594655E-002;
arCoef_Taps[5] := 	1.60017334206282E-002;
arCoef_Taps[6] := 	1.61369608038471E-002;
arCoef_Taps[7] := 	1.62672962073415E-002;
arCoef_Taps[8] :=	1.63926631245363E-002;
arCoef_Taps[9] :=	1.65129878977796E-002;
arCoef_Taps[10] :=	1.66281997700857E-002;

arCoef_Taps[11] :=  1.67382309348648E-002;
arCoef_Taps[12] :=  1.68430165836012E-002;
arCoef_Taps[13] :=  1.69424949514440E-002;
arCoef_Taps[14] :=  1.70366073606740E-002;
arCoef_Taps[15] :=  1.71252982620145E-002;
arCoef_Taps[16] :=  1.72085152737542E-002;
arCoef_Taps[17] :=  1.72862092186516E-002;
arCoef_Taps[18] :=  1.73583341585934E-002;
arCoef_Taps[19] :=  1.74248474269791E-002;
arCoef_Taps[20] :=  1.74857096588086E-002;

arCoef_Taps[21] :=  1.75408848184478E-002;
arCoef_Taps[22] :=  1.75903402250520E-002;
arCoef_Taps[23] :=  1.76340465756283E-002;
arCoef_Taps[24] :=  1.76719779657164E-002;
arCoef_Taps[25] :=  1.77041119076759E-002;
arCoef_Taps[26] :=  1.77304293465626E-002;
arCoef_Taps[27] :=  1.77509146735830E-002;
arCoef_Taps[28] :=  1.77655557371177E-002;
arCoef_Taps[29] :=  1.77743438513027E-002;
arCoef_Taps[30] :=  1.77772738021646E-002;

arCoef_Taps[31] :=  1.77743438513027E-002;
arCoef_Taps[32] :=  1.77655557371177E-002;
arCoef_Taps[33] :=  1.77509146735830E-002;
arCoef_Taps[34] :=  1.77304293465626E-002;
arCoef_Taps[35] :=  1.77041119076759E-002;
arCoef_Taps[36] :=  1.76719779657164E-002;
arCoef_Taps[37] :=  1.76340465756283E-002;
arCoef_Taps[38] :=  1.75903402250520E-002;
arCoef_Taps[39] :=  1.75408848184478E-002;
arCoef_Taps[40] :=  1.74857096588086E-002;

arCoef_Taps[41] :=  1.74248474269791E-002;
arCoef_Taps[42] :=  1.73583341585934E-002;
arCoef_Taps[43] :=  1.72862092186516E-002;
arCoef_Taps[44] :=  1.72085152737542E-002;
arCoef_Taps[45] :=  1.71252982620145E-002;
arCoef_Taps[46] :=  1.70366073606740E-002;
arCoef_Taps[47] :=  1.69424949514440E-002;
arCoef_Taps[48] :=  1.68430165836012E-002;
arCoef_Taps[49] :=  1.67382309348648E-002;
arCoef_Taps[50] :=  1.66281997700857E-002;

arCoef_Taps[51] :=  1.65129878977796E-002;
arCoef_Taps[52] :=  1.63926631245363E-002;
arCoef_Taps[53] :=  1.62672962073415E-002;
arCoef_Taps[54] :=  1.61369608038471E-002;
arCoef_Taps[55] :=  1.60017334206282E-002;
arCoef_Taps[56] :=  1.58616933594655E-002;
arCoef_Taps[57] :=  1.57169226616965E-002;
arCoef_Taps[58] :=  1.55675060506758E-002;
arCoef_Taps[59] :=  1.54135308723898E-002;


rSaida := 0.0;
FOR i:= 59 TO 2 BY -1 DO
	arLeitura[i] := arLeitura[i-1];	
	rAux := arLeitura[i] * arCoef_Taps[i];
	rSaida := rSaida + rAux;
END_FOR

arLeitura[1] := rEntrada;

rSaida := rSaida + (arLeitura[1] * arCoef_Taps[1]);

END_FUNCTION_BLOCK

// ---- POUs/FBs/P_TextModeWrite.TcPOU
(* Writing of CSV file in text mode. None of the field value is containing any non-printing control characters like line feed, carriage return, quotation marks, semicolon... *)
PROGRAM P_TextModeWrite
VAR
	bWrite			: BOOL := FALSE;(* Rising edge starts program execution *)
	sNetId			: T_AmsNetId := '';	(* TwinCAT system network address *)
	sFileName		: T_MaxString := 'C:\Temp\TextModeGen.csv';(* CSV destination file path and name *)
	sCSVLine		: T_MaxString := '';(* Single CSV text line (row, record), we are using string as record buffer (your are able to see created fields) *)
	sCSVField		: T_MaxString := '';(* Single CSV field value (column, record field) *)
	bBusy			: BOOL;
	bError			: BOOL;
	nErrId			: UDINT;
	nRow	 		: UDINT 	:= 0;(* Row number (record) *)
	nColumn			: UDINT 	:= 0;(* Column number (record field) *)
	hFile			: UINT		:= 0;(* File handle of the source file *)
	step			: DWORD 	:= 0;
	fbFileOpen		: FB_FileOpen;(* Opens file *)
	fbFileClose		: FB_FileClose;(* Closes file *)
	fbFilePuts		: FB_FilePuts;(* Writes one record (line) *)
	fbWriter		: FB_CSVMemBufferWriter;(* Helper function block used to create CSV data bytes (single record line) *)

	database		: ARRAY[0..MAX_CSV_ROWS, 0..MAX_CSV_COLUMNS ] OF STRING(MAX_CSV_FIELD_LENGTH) :=[ (* Source PLC database *)
	'0_0', '0_1', '0_2', '0_3', '0_4', '0_5',
	'1_0', '1_1', '1_2', '1_3', '1_4', '1_5',
	'2_0', '2_1', '2_2', '2_3', '2_4', '2_5',
	'3_0', '3_1', '3_2', '3_3', '3_4', '3_5',
	'4_0', '4_1', '4_2', '4_3', '4_4', '4_5',
	'5_0', '5_1', '5_2', '5_3', '5_4', '5_5'];

END_VAR

CASE step OF
	0:	(* Wait for rising edge at bWrite variable *)
		IF bWrite THEN
			bWrite 	:= FALSE;
			bBusy 	:= TRUE;
			bError	:= FALSE;
			nErrId	:= 0;
			hFile	:= 0;
			nRow	:= 0;
			nColumn	:= 0;
			step 	:= 1;
		END_IF

	1:	(* Open source file *)
		fbFileOpen(  bExecute := FALSE  );
		fbFileOpen( sNetId := sNetId, sPathName := sFileName, nMode := FOPEN_MODEWRITE OR FOPEN_MODETEXT,(* Open file in TEXT mode! *)
					ePath := PATH_GENERIC, bExecute := TRUE );
		step := 2;

	2:(* Wait until open not busy *)
		fbFileOpen( bExecute := FALSE, bError => bError, nErrID => nErrID, hFile => hFile );
		IF NOT fbFileOpen.bBusy THEN
			IF NOT fbFileOpen.bError THEN
				step := 3;
			ELSE(* Error: file not found? *)
				step := 100;
			END_IF
		END_IF

	3:(* Convert one PLC record to CSV format *)
		sCSVLine := '';
		fbWriter.eCmd := eEnumCmd_First;(* Write first field value *)
		IF nRow <= MAX_CSV_ROWS THEN

			FOR nColumn := 0 TO MAX_CSV_COLUMNS BY 1 DO

				sCSVField := STRING_TO_CSVFIELD( database[ nRow, nColumn ], FALSE );(* TODO: Get field value from your application *)

				(* Add new field to the record buffer *)
				fbWriter( 	pBuffer := ADR( sCSVLine ), cbBuffer := SIZEOF( sCSVLine ) - 1, putValue := sCSVField, pValue := 0, cbValue := 0,
							bCRLF := ( nColumn = MAX_CSV_COLUMNS ) );(* bCRLF == TRUE => Write CRLF after the last field value *)
				IF fbWriter.bOk THEN
					fbWriter.eCmd := eEnumCmd_Next;(* Write next field value *)
				ELSE(* Error *)
					step := 100;
					RETURN;
				END_IF

			END_FOR(* FOR nColumn := 0... *)

			(* FB_FilePuts adds allready CR (carriage return) to the written line.
			We have to replace the $R$L characters with $L character to avoid double CR. *)
			IF RIGHT( sCSVLine, 2 ) = '$R$L' THEN
				sCSVLine := REPLACE( sCSVLine, '$L', 2, LEN( sCSVLine ) - 1 );
			END_IF

			nRow := nRow + 1;(* Increment number of created records (rows) *)
			step := 4;(* Write record to the file *)

		ELSE(* All rows written => Close file *)
			step := 10;
		END_IF

	4:	(* Write single text line *)
		fbFilePuts( bExecute := FALSE );
		fbFilePuts( sNetId := sNetId, hFile := hFile, sLine := sCSVLine, bExecute := TRUE );
		step := 5;

	5:(* Wait until write not busy *)
		fbFilePuts( bExecute := FALSE, bError => bError, nErrID => nErrID );
		IF NOT fbFilePuts.bBusy THEN
			IF NOT fbFilePuts.bError THEN
				step := 3;(* Write next record *)
			ELSE(* Error *)
				step := 100;
			END_IF
		END_IF

	10:	(* Close source file *)
		fbFileClose( bExecute := FALSE );
		fbFileClose( sNetId := sNetId, hFile := hFile, bExecute := TRUE );
		step := 11;

	11:(* Wait until close not busy *)
		fbFileClose( bExecute := FALSE, bError => bError, nErrID => nErrID );
		IF ( NOT fbFileClose.bBusy ) THEN
			hFile := 0;
			step := 100;
		END_IF

	100: (* Error or ready step => cleanup *)
		IF ( hFile <> 0 ) THEN
			step := 10; (* Close the source file *)
		ELSE
			bBusy := FALSE;
			step := 0;	(* Ready *)
		END_IF

END_CASE

END_PROGRAM

// ---- POUs/FB_STATS.TcPOU
FUNCTION_BLOCK FB_STATS
VAR_INPUT
	bValidMeasurement		: BOOL;
	fLastWeight				: LREAL;
	fLastStd				: LREAL;
	bNewResult				: BOOL;
	bZerarGrafico			: BOOL;
	fReferenceMeasurement	: LREAL;
END_VAR
VAR_OUTPUT
	fMaxWeight				: LREAL;
	fMinWeight				: LREAL;
	fDelta					: LREAL;
	
	fMinReference			: LREAL;
	fMaxReference			: LREAL;
	fDeltaReference			: LREAL;
END_VAR
VAR
	arrGraph 			: ARRAY[1..1, 1..100] OF ST_POINTS;
	bSystemInit			: BOOL := FALSE;
	i					: INT;
	RTRIG_bNewResult		: R_TRIG;
	R_TRIG_bZerarGrafico	: R_TRIG;
	bFirstResult			: BOOL := TRUE;
	bCanRegister			: BOOL;
END_VAR

(* Last Weight Values to Plot in a Chart *)

IF NOT bSystemInit THEN
	(* Starting X reference chat *)
	FOR i:= 1 TO 100 DO
		arrGraph[1,i].x := i;
	END_FOR
END_IF

IF bValidMeasurement THEN
	(* Capture that we have Last Valid Weight until bNewResult Triggers *)
	bCanRegister	:= TRUE;
END_IF

RTRIG_bNewResult(CLK:= bCanRegister AND bNewResult, Q=> );

IF RTRIG_bNewResult.Q THEN
	(* FIFO for graph *)
	FOR i:= 100 TO 2 BY -1 DO
		arrGraph[1,i].y := arrGraph[1, i-1].y;
	END_FOR
	
	arrGraph[1,1].y 	:= fLastWeight;
	fLastWeight 		:= fLastWeight;
	fLastStd 			:= fLastStd;
	
	IF NOT bFirstResult THEN
		(* Check Max and Min Weighs *)
		IF fLastWeight > fMaxWeight THEN
			fMaxWeight := fLastWeight;
		END_IF
		
		IF fLastWeight < fMinWeight THEN
			fMinWeight := fLastWeight;
		END_IF
	ELSE
		fMaxWeight := fLastWeight;
		fMinWeight := fLastWeight;
		bFirstResult := FALSE;
	END_IF
	
	bCanRegister := FALSE;
END_IF

R_TRIG_bZerarGrafico(CLK:= bZerarGrafico, Q=> );

IF R_TRIG_bZerarGrafico.Q THEN
	FOR i:= 100 TO 1 BY -1 DO
		arrGraph[1,i].y := 0;
	END_FOR
	
	fMinWeight := 0;
	fMaxWeight := 0;
	bFirstResult := TRUE;
	fMinReference := 0;
	fMaxReference := 0;
END_IF

fDelta := fMaxWeight - fMinWeight;

(* Stats for Reference Signals [Raw or Filtered] Measurement *)

IF fMinReference = 0 THEN (* 0 means that no min value was registered *)
	fMinReference := fReferenceMeasurement;
ELSIF fReferenceMeasurement > fMaxReference THEN
	fMaxReference := fReferenceMeasurement;
	
ELSIF fReferenceMeasurement < fMinReference THEN
	fMinReference := fReferenceMeasurement;
END_IF

fDeltaReference := fMaxReference - fMinReference;

END_FUNCTION_BLOCK
